(* IEC 61131-3 sources: controlforge-structured-text/manual-tests/navigation, 5 files *)

(* ---- find-references.st ---- *)
(* Manual test: Find All References
   Right-click a symbol > "Find All References" (or Shift+F12).
   Verify all expected locations are listed in the References panel. *)

(* === Test 1: Variable with multiple references === *)
(* Find references on "counter" — expect declaration + 4 usages *)
PROGRAM FindRefsVarTest
VAR
    counter : INT := 0;
    max : INT := 100;
    done : BOOL;
END_VAR
    counter := counter + 1;
    IF counter >= max THEN
        done := TRUE;
        counter := 0;
    END_IF
END_PROGRAM

(* === Test 2: FB instance references including member access === *)
(* Find references on "myTimer" — expect declaration + all usages *)
PROGRAM FindRefsFBTest
VAR
    myTimer : TON;
    elapsed : BOOL;
END_VAR
    myTimer(IN := TRUE, PT := T#3s);
    elapsed := myTimer.Q;
END_PROGRAM

(* === Test 3: Variable with single reference === *)
(* Find references on "unused" — expect declaration only *)
PROGRAM FindRefsSingleTest
VAR
    unused : INT;
    used : INT;
END_VAR
    used := 42;
END_PROGRAM

(* === Test 4: Parameter in function block === *)
(* Find references on "enable" — expect declaration + body usage *)
FUNCTION_BLOCK FB_FindRefsTest
VAR_INPUT
    enable : BOOL;
    speed : REAL;
END_VAR
VAR_OUTPUT
    running : BOOL;
END_VAR
    running := enable AND (speed > 0.0);
END_FUNCTION_BLOCK

(* ---- member-access.st ---- *)
// Member Access Test File
// This file specifically tests function block member navigation
// Test cases for: instance.member → definition navigation

// Custom Function Block for testing
FUNCTION_BLOCK FB_MotorControl
VAR_INPUT
    start : BOOL;           // Start command
    stop : BOOL;            // Stop command
    speed : REAL;           // Desired speed (0-100%)
END_VAR
VAR_OUTPUT
    running : BOOL;         // Motor running status
    currentSpeed : REAL;    // Current actual speed
    fault : BOOL;           // Fault condition
END_VAR
VAR
    internalState : INT;    // Internal state machine
    rampTimer : TON;        // Speed ramping timer
END_VAR

// Simple motor control logic
IF start AND NOT stop THEN
    running := TRUE;
    currentSpeed := speed;
ELSIF stop THEN
    running := FALSE;
    currentSpeed := 0.0;
END_IF

// Ramp timer for smooth speed changes
rampTimer(IN := running, PT := T#2s);

END_FUNCTION_BLOCK

// Main test program
PROGRAM MemberAccessTest
VAR
    // Standard function block instances
    myTimer : TON;              // Timer instance
    edgeDetector : R_TRIG;      // Rising edge detector
    counter : CTU;              // Up counter

    // Custom function block instance
    motorCtrl : FB_MotorControl;  // Custom motor controller

    // Test variables
    enableSignal : BOOL;
    motorSpeed : REAL := 75.0;
    pulseSignal : BOOL;
    countValue : INT;
    timerDone : BOOL;
    motorStatus : BOOL;
    motorFault : BOOL;
END_VAR

// Test 1: Standard FB member access - Timer
// Navigate: myTimer.Q → should go to TON.Q definition
// Navigate: myTimer.PT → should go to TON.PT definition
myTimer(IN := enableSignal, PT := T#5s);
timerDone := myTimer.Q;        // Test navigation to .Q member
enableSignal := NOT myTimer.Q; // Test navigation to .Q member again

// Test 2: Standard FB member access - Edge detector
// Navigate: edgeDetector.CLK → should go to R_TRIG.CLK definition
// Navigate: edgeDetector.Q → should go to R_TRIG.Q definition
edgeDetector(CLK := pulseSignal);
IF edgeDetector.Q THEN         // Test navigation to .Q member
    countValue := countValue + 1;
END_IF

// Test 3: Standard FB member access - Counter
// Navigate: counter.CU → should go to CTU.CU definition
// Navigate: counter.CV → should go to CTU.CV definition
counter(CU := edgeDetector.Q, R := myTimer.Q, PV := 10);
countValue := counter.CV;      // Test navigation to .CV member

// Test 4: Custom FB member access
// Navigate: motorCtrl.start → should go to FB_MotorControl.start definition
// Navigate: motorCtrl.running → should go to FB_MotorControl.running definition
motorCtrl(
    start := enableSignal,     // Test navigation to .start member
    stop := FALSE,
    speed := motorSpeed        // Test navigation to .speed member
);

// Access output members
motorStatus := motorCtrl.running;  // Test navigation to .running member
motorFault := motorCtrl.fault;     // Test navigation to .fault member

// Test 5: Nested member access in expressions
IF (myTimer.Q AND motorCtrl.running) OR counter.Q THEN
    // Multiple member accesses in one expression
    // Navigate: myTimer.Q, motorCtrl.running, counter.Q
    motorSpeed := 50.0;
END_IF

// Test 6: Member access in function calls (future test case)
// This would be for when we implement function parameter navigation
// Example: SomeFunction(motorCtrl.currentSpeed, myTimer.ET);

END_PROGRAM

(* ---- peek-definition.st ---- *)
// Peek Definition (Alt+F12) — Manual QA Fixture
//
// HOW TO TEST
//   Open this file in VS Code with the extension active.
//   Press Alt+F12 on the indicated tokens to open the inline peek window.
//   Press Escape to close the peek window.
//   Press F12 to jump to the full definition instead.
//
// EXPECTED: peek window opens inline showing the definition source.
// EXPECTED: Escape closes the window without navigating.
// EXPECTED: F12 jumps to the definition file and closes the peek.

// ─── Custom symbols (cross-file peek) ────────────────────────────────────────

// Test 1: User-defined function block — peek shows FB_Counter body
FUNCTION_BLOCK FB_Counter
VAR_INPUT
    Enable : BOOL;
    Reset  : BOOL;
END_VAR
VAR_OUTPUT
    Count : INT;
    Done  : BOOL;
END_VAR
    IF Reset THEN
        Count := 0;
        Done  := FALSE;
    ELSIF Enable THEN
        Count := Count + 1;
        Done  := Count >= 10;
    END_IF;
END_FUNCTION_BLOCK

PROGRAM PeekTest
VAR
    // Alt+F12 on "FB_Counter" below — EXPECT: peek shows FUNCTION_BLOCK FB_Counter above (line 17)
    myCounter : FB_Counter;

    // Alt+F12 on "TON" below — EXPECT: peek opens iec61131-definitions/TON.st
    onDelay : TON;

    // Alt+F12 on "CTU" below — EXPECT: peek opens iec61131-definitions/CTU.st
    partCounter : CTU;

    // Alt+F12 on "R_TRIG" below — EXPECT: peek opens iec61131-definitions/R_TRIG.st
    risingEdge : R_TRIG;

    // Alt+F12 on "TOF" below — EXPECT: peek opens iec61131-definitions/TOF.st
    offDelay : TOF;

    // Alt+F12 on "TP" below — EXPECT: peek opens iec61131-definitions/TP.st
    pulse : TP;

    // Alt+F12 on "CTD" below — EXPECT: peek opens iec61131-definitions/CTD.st
    downCounter : CTD;

    // Alt+F12 on "CTUD" below — EXPECT: peek opens iec61131-definitions/CTUD.st
    biCounter : CTUD;

    // Alt+F12 on "F_TRIG" below — EXPECT: peek opens iec61131-definitions/F_TRIG.st
    fallingEdge : F_TRIG;

    // Alt+F12 on "RS" below — EXPECT: peek opens iec61131-definitions/RS.st
    resetDom : RS;

    // Alt+F12 on "SR" below — EXPECT: peek opens iec61131-definitions/SR.st
    setDom : SR;

    // Local variable — Alt+F12 on "Enable" below — EXPECT: peek shows VAR_INPUT Enable above (line 19)
    localEnable : BOOL;
END_VAR

// ─── Member access peek ────────────────────────────────────────────────────

onDelay(IN := localEnable, PT := T#3s);

// Alt+F12 on "onDelay" in "onDelay.Q" — EXPECT: peek shows instance declaration above
// Alt+F12 on "Q" in "onDelay.Q" — EXPECT: peek shows Q member in iec61131-definitions/TON.st
IF onDelay.Q THEN
    myCounter(Enable := TRUE, Reset := FALSE);
END_IF;

// Alt+F12 on "Count" in "myCounter.Count" — EXPECT: peek shows Count output in FB_Counter (line 25)
IF myCounter.Count >= 5 THEN
    localEnable := FALSE;
END_IF;

// ─── Multiple definitions (tabs in peek) ──────────────────────────────────

// Alt+F12 on "myCounter" — EXPECT: single peek location (the VAR declaration above)

END_PROGRAM

(* ---- local-vars.st ---- *)
// Quick test to verify local variable symbol indexing
PROGRAM TestLocalVars
VAR
    testTimer : TON;
    testCounter : CTU;
    localFlag : BOOL;
END_VAR

// Test navigation on these:
// 1. testTimer (should go to declaration)
// 2. testTimer.Q (should go to TON.Q member)
// 3. localFlag (should go to declaration)

testTimer(IN := TRUE, PT := T#1s);
localFlag := testTimer.Q;

END_PROGRAM

(* ---- navigation-targets.st ---- *)
// Test file to verify exact navigation targets
PROGRAM TestNavigation
VAR
    testTimer : TON;
END_VAR

// Navigate to these and verify the exact targets:
// 1. testTimer → should go to line 3 (local declaration)
// 2. testTimer.Q → should go to iec61131-definitions/TON.st line 9
// 3. testTimer.IN → should go to iec61131-definitions/TON.st line 5
// 4. testTimer.PT → should go to iec61131-definitions/TON.st line 6
// 5. testTimer.ET → should go to iec61131-definitions/TON.st line 10

testTimer(IN := TRUE, PT := T#5s);
IF testTimer.Q THEN
    // Timer has elapsed
END_IF

END_PROGRAM
